TYPE ST_AO :
STRUCT
		Value		  AT %Q*	: INT	;
		Description 			: STRING	;

END_STRUCT
END_TYPE

(* stored: Version 1.1.0.1, ProductVersion 3.1.4024.2
   DUT ST_AO: Id {afbf683e-d623-4191-a01d-e0767348f253} *)
